// Mitsubishi GX Works2 project: Project34_partB   PLC: FX3G

// global labels: Global1
VAR_GLOBAL
  StartAC AT X007 : BOOL;
  help0 AT M0 : BOOL;
  StopAC AT X010 : BOOL;
  ACon AT Y001 : BOOL;
  Temp25 AT X001 : BOOL;
  Timer1 AT TC1 : BOOL;
END_VAR
VAR_GLOBAL CONSTANT
  Time1 : INT := 50;
END_VAR
VAR_GLOBAL
  Timer1Output AT TS1 : BOOL;
END_VAR

// task Task_01 (event TRUE, interval 0, priority 31): POU_01

PROGRAM POU_01
(* structured ladder/FBD written out as ST: instructions are called as NAME(EN, inputs, outputs); _pN, _eN, _tN stand for wires *)
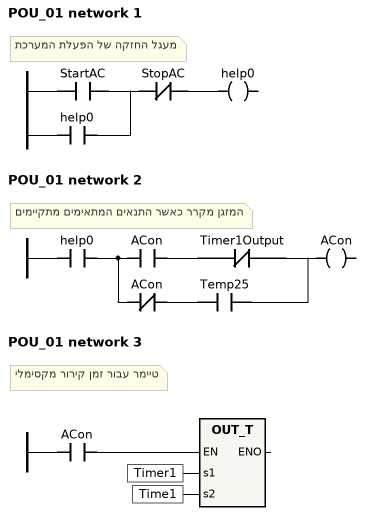
(* network 1 *)
(* מעגל החזקה של הפעלת המערכת *)
help0 := (StartAC OR help0) AND NOT StopAC;
(* network 2 *)
(* המזגן מקרר כאשר התנאים המתאימים מתקיימים *)
ACon := (help0 AND ACon AND NOT Timer1Output) OR (help0 AND NOT ACon AND Temp25);
(* network 3 *)
(* טיימר עבור זמן קירור מקסימלי *)
OUT_T(ACon, Timer1, Time1);
END_PROGRAM
